FUNCTION_BLOCK DigitalInput_NO EXTENDS Component IMPLEMENTS I_DigitalInput
VAR
	Input		  : REFERENCE TO BOOL;
	ForcibleInput : ForcibleBool(_Name);
END_VAR

//FB_Init is always available implicitly and it is used primarily for initialization.

//The return value is not evaluated. For a specific influence, you can also declare the

//methods explicitly and provide additional code there with the standard initialization

//code. You can evaluate the return value.
METHOD FB_Init : BOOL
VAR_INPUT
	bInitRetains : BOOL; // TRUE: the retain variables are initialized (reset warm / reset cold)
	bInCopyCode	 : BOOL; // TRUE: the instance will be copied to the copy code afterward (online change)   
	Name		 : T_MaxString;
	Input		 : REFERENCE TO BOOL;
END_VAR
THIS^.Input REF= Input;
END_METHOD

{attribute 'monitoring' := 'call'}
PROPERTY Force : E_ForceState
GET
Force := ForcibleInput.CurrentForceState;
END_GET
SET
VAR
	ForceString : T_MaxString := TO_STRING(Force);
END_VAR
ForcibleInput.SetForceState(Force);
END_SET
END_PROPERTY

{attribute 'monitoring' := 'call'}
PROPERTY IsActive : BOOL
GET
ForcibleInput.Input := Input;
IsActive			:= ForcibleInput.Output;
END_GET
END_PROPERTY

END_FUNCTION_BLOCK

(* stored: Version 1.1.0.1, ProductVersion 3.1.4026.18
   POU DigitalInput_NO: Id {9d9dda3a-7e57-4cae-a0d6-f476ce62c0a0}, SpecialFunc None
   Method FB_Init: Id {a130aac5-6f41-4a7d-9b06-f9d6875f364c}
   Property Force: Id {c17864b9-2486-420f-bbaf-a2f4879fb828}
   Get Get: Id {91f3c0ff-d2ee-44c7-9f3c-bda3f96e031c}
   Set Set: Id {84a591c0-696f-4881-932f-68c716bb0db3}
   Property IsActive: Id {ab760981-4737-4823-a793-9cafc734e1c9}
   Get Get: Id {2bb650fa-fe8b-42cc-aed4-245829767bd1} *)
